(* CoDeSys 2.3.9.35 project: washing_machine.pro *)
(* Author: Altus *)
(* Libraries: DU35x.lib 7.7.11 15:59:13, Navigation.lib 15.7.11 10:06:00, SysLibTargetVisu.lib 26.11.08 09:53:28, Standard.lib 26.11.08 09:46:20, Iecsfc.lib 26.11.08 09:46:14, SYSLIBCALLBACK.LIB 26.11.08 09:53:30 *)

(* PLC configuration (modules and I/O channels)
MToolIEC [Codesys] node 0, in %IB0 out %QB0
Desabilitada [Desabilitado485] node 0, in %IB0 out %QB0
Entradas Digitais 0 [Entradas0] node 0, in %IW0 out %QB0
  I00 AT %IX0.0 [BitInput] I0.0
  I01 AT %IX0.1 [BitInput] I0.1
  I02 AT %IX0.2 [BitInput] I0.2
  I03 AT %IX0.3 [BitInput] I0.3
  I04 AT %IX0.4 [BitInput] I0.4
  I05 AT %IX0.5 [BitInput] I0.5
  I06 AT %IX0.6 [BitInput] I0.6
  I07 AT %IX0.7 [BitInput] I0.7
  I08 AT %IX0.8 [BitInput] I0.8
Entradas Digitais 1 [Entradas1] node 0, in %IW1 out %QB0
  I10 AT %IX1.0 [BitInput] I1.0
  I11 AT %IX1.1 [BitInput] I1.1
  I12 AT %IX1.2 [BitInput] I1.2
  I13 AT %IX1.3 [BitInput] I1.3
  I14 AT %IX1.4 [BitInput] I1.4
  I15 AT %IX1.5 [BitInput] I1.5
  I16 AT %IX1.6 [BitInput] I1.6
  I17 AT %IX1.7 [BitInput] I1.7
  I18 AT %IX1.8 [BitInput] I1.8
Entradas Digitais 2 [Entradas2] node 0, in %IW2 out %QB0
  I20 AT %IX2.0 [BitInput] I2.0
  I21 AT %IX2.1 [BitInput] I2.1
Entradas Analógicas [EntradaAnalogica] node 0, in %IW4 out %QB0
  AI0 AT %IW4 [WordInput] AI0 {TipoAnalogica = Tensão 0-10V; FiltroAnalogica = Filtro 0 - AI=2ms  / AV=90ms; FundoEscala = 100}
  AI1 AT %IW5 [WordInput] AI1 {TipoAnalogica = Canal Desabilitado; FiltroAnalogica = Filtro 0 - AI=2ms  / AV=90ms; FundoEscala = 0}
  AI2 AT %IW6 [WordInput] AI2 {TipoAnalogica = Canal Desabilitado; FiltroAnalogica = Filtro 0 - AI=2ms  / AV=90ms; FundoEscala = 0}
  AI3 AT %IW7 [WordInput] AI3 {TipoAnalogica = Canal Desabilitado; FiltroAnalogica = Filtro 0 - AI=2ms  / AV=90ms; FundoEscala = 0}
Entradas Rápidas [EntradasRapidas] node 1, in %IB16 out %QB0
  Bloco 0 [Bloco0] node 0, in %IB16 out %QB0
    Desabilitado [DesabilitadoBloco0] node 0, in %IB16 out %QB0
  Bloco 1 [Bloco1] node 1, in %IB16 out %QB0
    Desabilitado [DesabilitadoBloco1] node 0, in %IB16 out %QB0
  Entrada Configuravél Bloco 0 [EntradaConfiBloco0] node 2, in %IB16 out %QB0
    Contador 0 [EntradaConfContador0] node 0, in %IB16 out %QB0 {EntradaConfiguravelContador = Disable}
  Entrada Configuravél Bloco 1 [EntradaConfiBloco1] node 3, in %IB16 out %QB0
    Contador 2 [EntradaConfContador2] node 0, in %IB16 out %QB0 {EntradaConfiguravelContador = Disable}
Saídas Digitais 0 [Saidas0] node 0, in %IW0 out %QW0
  Q00 AT %QX0.0 [BitOutput] Q0.0
  Q01 AT %QX0.1 [BitOutput] Q0.1
  Q02 AT %QX0.2 [BitOutput] Q0.2
  Q03 AT %QX0.3 [BitOutput] Q0.3
  Q04 AT %QX0.4 [BitOutput] Q0.4
  Q05 AT %QX0.5 [BitOutput] Q0.5
  Q06 AT %QX0.6 [BitOutput] Q0.6
  Q07 AT %QX0.7 [BitOutput] Q0.7
Saídas Digitais 1 [Saidas1] node 0, in %IW0 out %QW1
  Q10 AT %QX1.0 [BitOutput] Q1.0
  Q11 AT %QX1.1 [BitOutput] Q1.1
  Q12 AT %QX1.2 [BitOutput] Q1.2
  Q13 AT %QX1.3 [BitOutput] Q1.3
  Q14 AT %QX1.4 [BitOutput] Q1.4
  Q15 AT %QX1.5 [BitOutput] Q1.5
  Q16 AT %QX1.6 [BitOutput] Q1.6
  Q17 AT %QX1.7 [BitOutput] Q1.7
AO0 AT %QW3 [WordOutput] AO0 {TipoAnalogica = Canal Desabilitado; FundoEscala = 0}
AO1 AT %QW4 [WordOutput] AO1 {TipoAnalogica = Canal Desabilitado; FundoEscala = 0}
Saída Rápida 0 Desabilitada [DesabilitadoF0] node 0, in %IB0 out %QB10
PTO [PTOF1] node 1, in %IB0 out %QB10 {RampaPTO = Trapezoidal}
Saídas Comum de Contador [SaidasContador] node 2, in %IB0 out %QB10
  Saída do Bloco 0 Desabilitada [DesabilitadoSaidaBloco0] node 0, in %IB0 out %QB10
  Saída do Bloco 1 Desabilitada [DesabilitadoSaidaBloco1] node 1, in %IB0 out %QB10
Evento Temporizado [TimerEvent] node 0, in %IB13 out %QB6 {Intervalo = 10}
*)

(* Task configuration *)
TASK PRINCIPAL (PRIORITY := 1, INTERVAL := T#1ms);
	PLC_PRG();
END_TASK
TASK NAVIGATION (PRIORITY := 1, INTERVAL := T#20ms);
	NAVEGA();
END_TASK
TASK VISUALIZATION (PRIORITY := 1, INTERVAL := T#500ms);
	MAINTARGETVISU_PAINT_CODE
END_TASK
TASK KEYBOARD_USAGE (PRIORITY := 1, INTERVAL := T#20ms);
	MAINTARGETVISU_INPUT_CODE
END_TASK

(* POU PLC_PRG, LD *)
PROGRAM PLC_PRG
VAR

	FREQ AT %MD1652: DWORD :=0;
	PULSOS AT %MD1653: DWORD :=0;
	RAMPA AT %MD1654: DWORD :=0;
	SENTIDO AT %QX0.2: BOOL := 0;
	START AT %MX3314.2: BOOL :=0;
	STOP AT %MX3314.3: BOOL :=0;

	NORMAL: BOOL;
	RAPIDO: BOOL;
	TURBO: BOOL;

	CONDICAO: CondicaoModo;
	MODO: STRING;

END_VAR
VAR_INPUT

	LIGAR AT %IX0.0: BOOL := 0;
	DESLIGAR AT %IX0.1: BOOL := 0;
	Mudar_sentido AT %IX0.5: BOOL := 0;
	VEL1 AT %IX0.2: BOOL := 0;
	VEL2 AT %IX0.3: BOOL := 0;
	VEL3 AT %IX0.4: BOOL := 0;
	POT AT %IW4: WORD := 0;

END_VAR
VAR_OUTPUT

	SIST AT %QX1.0: BOOL;

END_VAR
VAR (* helpers for the ST form of the networks *)
	_p1 : BOOL;
	_p2 : BOOL;
END_VAR
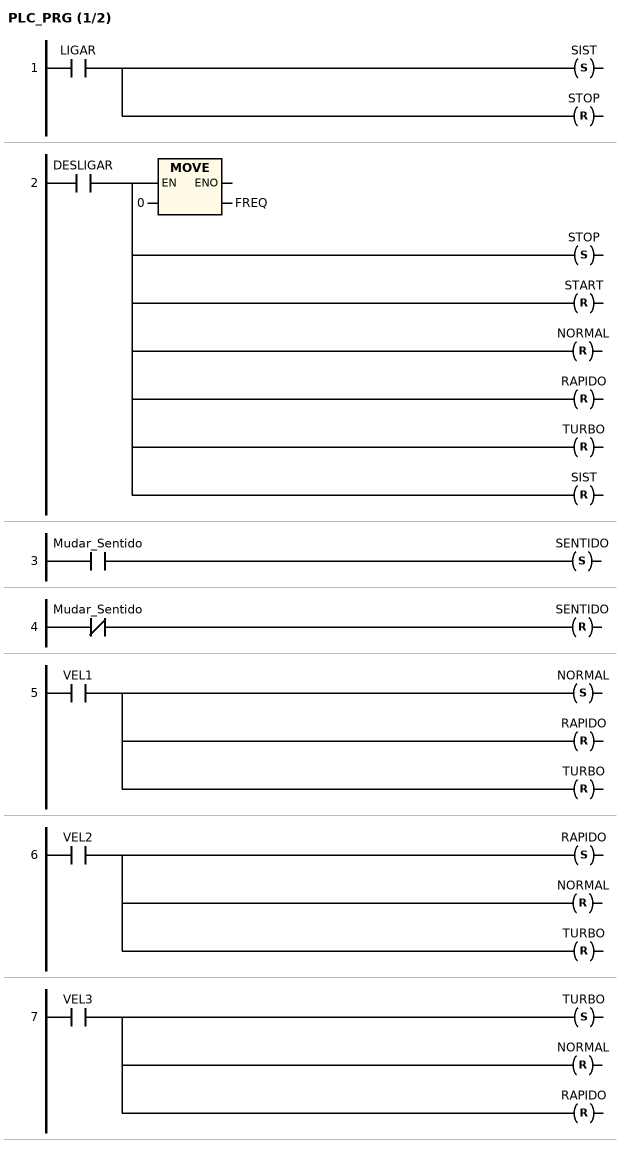
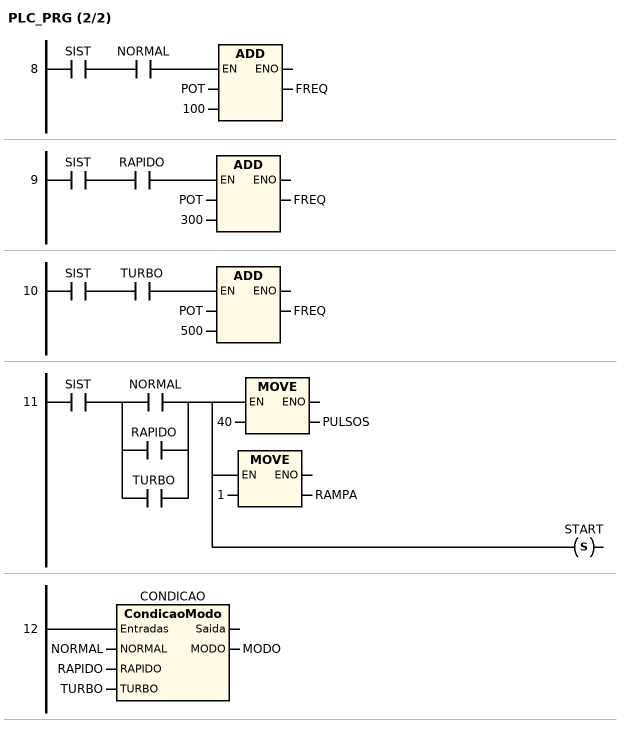
_LD_ (* Ladder Diagram *)
NETWORK 1
	[LIGAR] --- (S SIST) (R STOP)
NETWORK 2
	[DESLIGAR] --- (S STOP) (R START) (R NORMAL) (R RAPIDO) (R TURBO) (R SIST)
		EN --- MOVE(0) => FREQ
NETWORK 3
	[Mudar_Sentido] --- (S SENTIDO)
NETWORK 4
	[/Mudar_Sentido] --- (R SENTIDO)
NETWORK 5
	[VEL1] --- (S NORMAL) (R RAPIDO) (R TURBO)
NETWORK 6
	[VEL2] --- (S RAPIDO) (R NORMAL) (R TURBO)
NETWORK 7
	[VEL3] --- (S TURBO) (R NORMAL) (R RAPIDO)
NETWORK 8
	[SIST] - [NORMAL]
		EN --- ADD(POT, 100) => FREQ
NETWORK 9
	[SIST] - [RAPIDO]
		EN --- ADD(POT, 300) => FREQ
NETWORK 10
	[SIST] - [TURBO]
		EN --- ADD(POT, 500) => FREQ
NETWORK 11
	[SIST] - { [NORMAL] | [RAPIDO] | [TURBO] } --- (S START)
		EN --- MOVE(40) => PULSOS
		EN --- MOVE(1) => RAMPA
NETWORK 12
	CONDICAO:CondicaoModo(Entradas: *, NORMAL: NORMAL, RAPIDO: RAPIDO, TURBO: TURBO, MODO => MODO)
_END_LD_
(* the same logic as Structured Text *)
(* Network 1 *)
IF LIGAR THEN SIST := TRUE; STOP := FALSE; END_IF;
(* Network 2 *)
_p1 := DESLIGAR;
IF _p1 THEN
	FREQ := 0;
END_IF;
IF _p1 THEN STOP := TRUE; START := FALSE; NORMAL := FALSE; RAPIDO := FALSE; TURBO := FALSE; SIST := FALSE; END_IF;
(* Network 3 *)
IF Mudar_Sentido THEN SENTIDO := TRUE; END_IF;
(* Network 4 *)
IF NOT Mudar_Sentido THEN SENTIDO := FALSE; END_IF;
(* Network 5 *)
IF VEL1 THEN NORMAL := TRUE; RAPIDO := FALSE; TURBO := FALSE; END_IF;
(* Network 6 *)
IF VEL2 THEN RAPIDO := TRUE; NORMAL := FALSE; TURBO := FALSE; END_IF;
(* Network 7 *)
IF VEL3 THEN TURBO := TRUE; NORMAL := FALSE; RAPIDO := FALSE; END_IF;
(* Network 8 *)
IF SIST AND NORMAL THEN
	FREQ := POT + 100;
END_IF;
(* Network 9 *)
IF SIST AND RAPIDO THEN
	FREQ := POT + 300;
END_IF;
(* Network 10 *)
IF SIST AND TURBO THEN
	FREQ := POT + 500;
END_IF;
(* Network 11 *)
_p2 := SIST AND (NORMAL OR RAPIDO OR TURBO);
IF _p2 THEN
	PULSOS := 40;
	RAMPA := 1;
END_IF;
IF _p2 THEN START := TRUE; END_IF;
(* Network 12 *)
CONDICAO(Entradas := TRUE, NORMAL := NORMAL, RAPIDO := RAPIDO, TURBO := TURBO);
MODO := CONDICAO.MODO;
END_PROGRAM

(* POU CondicaoModo, ST *)
FUNCTION_BLOCK CondicaoModo
VAR_INPUT
	Entradas: BOOL;
	NORMAL: BOOL;
	RAPIDO: BOOL;
	TURBO: BOOL;
END_VAR
VAR_OUTPUT
	Saida: BOOL;
	MODO: STRING;
END_VAR
VAR
END_VAR
IF NORMAL=1 THEN MODO := 'normal';
ELSIF RAPIDO=1 THEN MODO := 'rapido';
ELSIF TURBO=1 THEN MODO := 'turbo';
ELSE MODO := 'parado';
END_IF
END_FUNCTION_BLOCK

(* POU NAVEGA, ST *)
PROGRAM NAVEGA
VAR
	ControleTelas : NAVIGATION;
	ListaTelas 	: ARRAY [0..30] OF STRING(10);
END_VAR
(* Adiciona a tela MAIN como tela principal *)
ListaTelas[0] := 'MAIN';

(* Ativa o controle automático de navegação somente pelo teclado *)
ControleTelas(ENABLE_UPDW := FALSE, VISU_LIST := ListaTelas, UP := FALSE , DOWN := FALSE);
END_PROGRAM

(* Visualisation MAIN
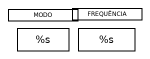
rectangle at (67,23)-(124,46): text "%s"; shows PLC_PRG.FREQ
rectangle at (61,3)-(131,15): text "FREQUÊNCIA"
rectangle at (6,23)-(58,46): text "%s"; shows PLC_PRG.MODO
rectangle at (-3,4)-(67,16): text "MODO"
*)
